// TIA Portal V19 export
DATA_BLOCK "Straightener"   // DB65
// stored: InstanceOfName Straightener_FB, InstanceOfType FB
"Straightener_FB"
   // VAR_INPUT
   //    AreaInterface : "AreaInterface";
   //    ZSI : "udt_ZoneSafetyInterface";
   //    DSI : Struct
   //       Feed : "udt_DeviceSafetyInterface";
   //       Lift_Entry : "udt_DeviceSafetyInterface";
   //       Lift_Exit : "udt_DeviceSafetyInterface";
   //    END_STRUCT;
   //    Drive : Struct
   //       Feed : "TAx_DriveInterface";
   //    END_STRUCT;
   //    DataIn : Struct
   //       Feed : "PositioningMachine_DataIn";
   //       Lift_Entry : "ValveMachine_DataIn";
   //       Lift_Exit : "ValveMachine_DataIn";
   //    END_STRUCT;
   //    CIn : Struct
   //       Manager : "Straightener_Manager";
   //       Feed_BwdEnable : Array[1..8] of Bool;
   //       Feed_FwdEnable : Array[1..8] of Bool;
   //    END_STRUCT;
   //    Config : Struct
   //       Feed : "PositioningMachine_Config";
   //       Lift_Entry : "ValveMachine_Config";
   //       Lift_Exit : "ValveMachine_Config";
   //       Lift_Entry_Exist : Bool;
   //       Lift_Exit_Exist : Bool;
   //    END_STRUCT;
   // END_VAR
   // VAR_OUTPUT
   //    MachineInterface : "MachineInterface";
   //    DataOut : Struct
   //       Feed : "PositioningMachine_DataOut";
   //       Lift_Entry : "ValveMachine_DataOut";
   //       Lift_Exit : "ValveMachine_DataOut";
   //    END_STRUCT;
   //    COut : "Straightener_Status";
   // END_VAR
   // VAR_IN_OUT
   //    TO_Ax : TO_PositioningAxis;
   //    PersistentValues : Struct
   //       Data : Struct
   //          Feed : "PositioningMachine_DataPers";
   //       END_STRUCT;
   //       Feed : "PositioningMachine_Par";
   //    END_STRUCT;
   // END_VAR
   // VAR
   //    Alarm : Struct
   //       Feed : "PositioningMachine_Alr";
   //       Lift_Entry : "ValveAlr";
   //       Lift_Exit : "ValveAlr";
   //    END_STRUCT;
   //    Warning : Struct
   //       Feed : "PositioningMachine_Wng";
   //       Lift_Entry : "ValveMachine_Wng";
   //       Lift_Exit : "ValveMachine_Wng";
   //    END_STRUCT;
   //    Feed : "PositioningMachine_FB";
   //    Lift_Entry : "ValveMachine_FB";
   //    Lift_Exit : "ValveMachine_FB";
   // END_VAR
BEGIN
END_DATA_BLOCK
